(*
:Class for handling communications between a client requesting a service 
:and a server providing the service
*)
{attribute 'reflection'}
FUNCTION_BLOCK T_Execution IMPLEMENTS I_Execution
VAR
    _State   : T_ExecutionState;
    _Done    : BOOL;
    _Error   : BOOL;
    _Aborted : BOOL;
    _ErrorMsg : T_MaxString;

    {attribute 'instance-path'} {attribute 'no_init'}
    Name : T_MaxString; // Automatically initialised with the full name of the instance

    _Notification_OnError : I_Notification;
    _Notification_OnAbort : I_Notification;
END_VAR

METHOD Abort
VAR_INPUT
END_VAR
// Aborting must be handled by the client class - cleanup and set Ready state
IF NOT _Aborted THEN // avoid going back into borting if execution has already been aborted
    _State := T_ExecutionState.Aborting; 
END_IF
END_METHOD

PROPERTY Aborted : BOOL
GET
Aborted := _Aborted;
END_GET
END_PROPERTY

PROPERTY Aborting : BOOL
GET
Aborting := _State = T_ExecutionState.Aborting;
END_GET
END_PROPERTY

PROPERTY Busy : BOOL
GET
Busy := _State = T_ExecutionState.Busy;
END_GET
END_PROPERTY

// Clears the results flags provided State = Ready
METHOD Clear
IF _State = T_ExecutionState.Ready THEN
    _Done     := FALSE;
    _Aborted  := FALSE;
    _Error    := FALSE;
    _ErrorMsg := '';
ELSE
    IF _Notification_OnError <> 0 THEN
        _Notification_OnError.Args
            .Clear()
            .Add_STRING('Clear requested while not ready')
            .Add_STRING(Name);

        _Notification_OnError.Raise();
    END_IF
END_IF
END_METHOD

PROPERTY Done : BOOL
GET
Done := _Done;
END_GET
END_PROPERTY

PROPERTY Error : BOOL
GET
Error := _Error;
END_GET
END_PROPERTY

PROPERTY ErrorMsg : T_MaxString
GET
ErrorMsg := _ErrorMsg;
END_GET
END_PROPERTY

// Individual T_Execution events are assigned here to the global events 
// so by default, all errors/aborts raise these global events
// This can be overidden for individual instances or T_Execution 
// by setting the Event properties to zero (or another event)
METHOD FB_init : BOOL
VAR_INPUT
	bInitRetains : BOOL; // if TRUE, the retain variables are initialized (warm start / cold start)
	bInCopyCode : BOOL;  // if TRUE, the instance afterwards gets moved into the copy code (online change)
END_VAR
_Notification_OnAbort := GlobalNotifications.Notification_ExecutionAborted;
_Notification_OnError := GlobalNotifications.Notification_ExecutionFailed;
END_METHOD

PROPERTY Notification_OnAbort : I_Notification
GET
Notification_OnAbort := _Notification_OnAbort;
END_GET
SET
_Notification_OnAbort := Notification_OnAbort;
END_SET
END_PROPERTY

PROPERTY Notification_OnError : I_Notification
GET
Notification_OnError := _Notification_OnError;
END_GET
SET
_Notification_OnError := Notification_OnError;
END_SET
END_PROPERTY

PROPERTY Ready : BOOL
GET
Ready := _State = T_ExecutionState.Ready;
END_GET
END_PROPERTY

METHOD SetAborted // used when implementing class signals Aborted
IF _State = T_ExecutionState.Starting OR _State = T_ExecutionState.Busy THEN
    _Aborted := TRUE;
    _State := T_ExecutionState.Ready;
    
    IF _Notification_OnAbort <> 0 THEN
        _Notification_OnAbort.Args.Add_STRING(F_FormatString1('Execution aborted in %s',F_STRING(Name)));
        _Notification_OnAbort.Raise();
    END_IF  

END_IF

IF _State = T_ExecutionState.Aborting THEN
    _Done     := FALSE;
    _Aborted  := TRUE;
    _Error    := FALSE;
    _ErrorMsg := 'Aborted';

    _State := T_ExecutionState.Ready;
END_IF
END_METHOD

METHOD SetBusy
VAR_INPUT
END_VAR
IF _State = T_ExecutionState.Starting THEN
    _State := T_ExecutionState.Busy;
END_IF
END_METHOD

METHOD SetDone
VAR_INPUT
END_VAR
IF _State = T_ExecutionState.Starting OR _State = T_ExecutionState.Busy THEN
    _Error    := FALSE;
    _ErrorMsg := '';
    _Aborted  := FALSE;
    _Done     := TRUE;
    _State    := T_ExecutionState.Ready;
END_IF
END_METHOD

METHOD SetError
VAR_INPUT
    ErrorMsg  : T_MaxString;
END_VAR
VAR
	pSTRING : POINTER TO STRING;
	arg : T_Arg;
END_VAR
IF _State = T_ExecutionState.Starting OR _State = T_ExecutionState.Busy THEN
    _Error    := TRUE;
    _Aborted  := FALSE;
    _Done     := FALSE;
    _ErrorMsg := ErrorMsg;
    _State    := T_ExecutionState.Ready;

    IF _Notification_OnError <> 0 THEN
        _Notification_OnError.Args
            .Clear()
            .Add_STRING(_ErrorMsg)
            .Add_STRING(Name);

        _Notification_OnError.Raise();
    END_IF

END_IF
END_METHOD

METHOD Start : BOOL
VAR_INPUT
END_VAR
IF _State = T_ExecutionState.Ready THEN
    _Done     := FALSE;
    _Aborted  := FALSE;
    _Error    := FALSE;
    _ErrorMsg := '';

    _State := T_ExecutionState.Starting;
    Start  := TRUE; // Accepted
ELSE
    IF _Notification_OnError <> 0 THEN
        _Notification_OnError.Args
            .Clear()
            .Add_STRING('Start requested while not ready')
            .Add_STRING(Name);

        _Notification_OnError.Raise();
    END_IF
END_IF
END_METHOD

PROPERTY Starting : BOOL
GET
Starting := _State = T_ExecutionState.Starting;
END_GET
END_PROPERTY

PROPERTY State : T_ExecutionState
GET
State := _State;
END_GET
END_PROPERTY

END_FUNCTION_BLOCK

(* stored: Version 1.1.0.1, ProductVersion 3.1.4024.9
   POU T_Execution: Id {b17395d1-e10b-079c-263b-2eb9c4f6194b}, SpecialFunc None
   Folder Methods: Id {e45bf685-06c9-4e29-a8a9-cbf0453f59ad}
   Folder Properties: Id {a48b7191-6aa5-4ac4-bdc5-b99d3da36639}
   Method Abort: Id {f3b9b616-ecb6-448b-9a68-cf8864d1ed1d}
   Property Aborted: Id {47f18dce-47db-4b5b-a019-8668343f98f9}
   Get Get: Id {f0f7563d-0a03-015d-3c7f-c1748808105b}
   Property Aborting: Id {f8431846-1954-03c8-30df-5a7e741c3ebe}
   Get Get: Id {eb3b9983-c850-041a-1155-83f5216a49d2}
   Property Busy: Id {03e849ec-ee28-0870-1ae9-eeb1ed24f4bc}
   Get Get: Id {945a4888-d71c-0d67-2d11-1ee4fe1836ec}
   Method Clear: Id {e820ac7a-e3e5-421e-9394-79fc023e1ef0}
   Property Done: Id {b9177cfb-6140-0c22-2370-60610db97e0d}
   Get Get: Id {bc67d8cf-9e35-059a-2bc9-46701e812750}
   Property Error: Id {4a58af1f-20ba-01b9-3bbb-3123d27f16d2}
   Get Get: Id {1bbb2e91-5896-0439-3898-15f12447c831}
   Property ErrorMsg: Id {03b333cf-212f-4b26-bcfc-f54366a3390d}
   Get Get: Id {87c8799e-98ff-4462-b8ed-e28804a16aed}
   Method FB_init: Id {cb8c0a25-6839-0ca3-105e-335fcd806bf2}
   Property Notification_OnAbort: Id {0d67ae06-841f-4128-bead-022f0ca9e3d9}
   Get Get: Id {03dd9ffc-038b-436c-8c4b-b9b9ae4aa681}
   Set Set: Id {2d2b3777-2c06-46db-b1c9-854dc3714dd4}
   Property Notification_OnError: Id {38d0423b-9d60-41ef-adab-a0253263c4b6}
   Get Get: Id {7560c815-0306-43f8-ac55-87c1998d7e74}
   Set Set: Id {228f6cfe-d91d-4d86-8b07-6069ae0ee2a8}
   Property Ready: Id {2af7d30b-7188-0edf-32b7-9305dcd7f6c3}
   Get Get: Id {07819190-be5b-06a7-0f77-77e004f7eaea}
   Method SetAborted: Id {3457d55d-8917-427f-b4b1-3d8dae8fe5f2}
   Method SetBusy: Id {a5a7c695-c8c2-0fa3-058b-7078b33d95e5}
   Method SetDone: Id {7437ab2d-de97-0db9-2d0a-b86eae15da44}
   Method SetError: Id {f1633771-a524-4ccc-be65-99229396429e}
   Method Start: Id {def3bafe-9648-0b74-364e-7150751f5a3a}
   Property Starting: Id {74926035-220d-03e3-3b86-d5067a70c227}
   Get Get: Id {b249388e-1ee2-027a-08c8-85eee11e571e}
   Property State: Id {34686f20-e5ce-076a-20fe-0604181ce5eb}
   Get Get: Id {643951a8-dea2-0da6-338f-29e7e986b3be} *)
